Staubli VAL3: Staubli.dtx

public SetDrivePwrMsg setDrvPwrAck
  [0]
    bool bDrivePower
    Body body
      [0]
        num nData
    Header header
      [0]
        num nCommType
        num nData[12]
        num nMsgType
        num nReplyCode
    Prefix prefix
      [0]
        num nData[4]
        num nLength
public SetDrivePwrMsg setDrvPwrMsg
  [0]
    bool bDrivePower
    Body body
      [0]
        num nData
    Header header
      [0]
        num nCommType
        num nData[12]
        num nMsgType
        num nReplyCode
    Prefix prefix
      [0]
        num nData[4]
        num nLength
public VelocityCfgMsg velCfgAck
  [0]
    Body body
      [0]
        num nData[68]
    Header header
      [0]
        num nCommType
        num nData[12]
        num nMsgType
        num nReplyCode
    Prefix prefix
      [0]
        num nData[4]
        num nLength = 76
    VelocityCfg velCfg
      [0]
        num nAccel
        num nCmdType
        num nRefFrameVec[6]
        num nRotVel
        num nToolVec[6]
        num nTransVel
public VelocityCfgMsg velCfgMsg
  [0]
    Body body
      [0]
        num nData[68]
    Header header
      [0]
        num nCommType
        num nData[12]
        num nMsgType
        num nReplyCode
    Prefix prefix
      [0]
        num nData[4]
        num nLength
    VelocityCfg velCfg
      [0]
        num nAccel
        num nCmdType
        num nRefFrameVec[6]
        num nRotVel
        num nToolVec[6]
        num nTransVel
public VelocityCmdMsg velCmdAck
  [0]
    Body body
      [0]
        num nData[32]
    Header header
      [0]
        num nCommType
        num nData[12]
        num nMsgType
        num nReplyCode
    Prefix prefix
      [0]
        num nData[4]
        num nLength = 44
    VelocityCmd velCmd
      [0]
        num nCmdType
        num nSeq
        num nVelVec[6]
public VelocityCmdMsg velCmdMsg
  [0]
    Body body
      [0]
        num nData[32]
    Header header
      [0]
        num nCommType
        num nData[12]
        num nMsgType
        num nReplyCode
    Prefix prefix
      [0]
        num nData[4]
        num nLength
    VelocityCmd velCmd
      [0]
        num nCmdType
        num nSeq
        num nVelVec[6]
public WriteSingIOMsg writeSingIOMsg
  [0]
    Body body
      [0]
        num nData[9]
    Header header
      [0]
        num nCommType
        num nData[12]
        num nMsgType
        num nReplyCode
    Prefix prefix
      [0]
        num nData[4]
        num nLength
    WriteSingleIO writeSingleIO
      [0]
        bool bState
        num nModuleId
        num nPin
public WriteSingIOMsg writeSingIOAck
  [0]
    Body body
      [0]
        num nData[9]
    Header header
      [0]
        num nCommType
        num nData[12]
        num nMsgType
        num nReplyCode
    Prefix prefix
      [0]
        num nData[4]
        num nLength
    WriteSingleIO writeSingleIO
      [0]
        bool bState
        num nModuleId
        num nPin
public _MotionMode MotionMode
  [0]
    num INVALID
    num JOINT_TRAJ = 1
    num VELOCITY_CTRL = 4
public _MsgTypeStaubli MsgType
  [0]
    num SET_DRIVE_POWER
    num VELOCITY_CFG = 1640
    num VELOCITY_CMD = 1641
    num READ_IO
    num WRITE_SINGLE_IO
public _VelocityType VelocityType
  [0]
    num INVALID
    num JOINT = 1
    num BASE_FRAME = 2
    num TOOL_FRAME = 3
